// EN: Endpoint flags depend on actual feedback and remain valid
//     independently of the active automatic target.
// PT: As flags de extremidade dependem do feedback real e permanecem
//     válidas independentemente do alvo automático ativo.
elevatorAtMinPosition :=
    elevatorHomed AND
    (
        elevatorLowerLimit OR
        (
            elevatorPositionMm <=
            (
                machineConfig.elevatorMinPositionMm +
                MAX(0.0, machineConfig.elevatorPositionToleranceMm)
            )
        )
    );

elevatorAtMaxPosition :=
    elevatorHomed AND
    (
        elevatorUpperLimit OR
        (
            elevatorPositionMm >=
            (
                machineConfig.elevatorMaxPositionMm -
                MAX(0.0, machineConfig.elevatorPositionToleranceMm)
            )
        )
    );

elevatorInPosition :=
    elevatorHomed AND
    (
        (elevatorAbsPositionErrorMm <= machineConfig.elevatorPositionToleranceMm)
        OR
        (
            elevatorUpperLimit AND
            (elevatorTargetPositionMm >= machineConfig.elevatorMaxPositionMm)
        )
        OR
        (
            elevatorLowerLimit AND
            (elevatorTargetPositionMm <= machineConfig.elevatorMinPositionMm)
        )
    );


//==============================================================
// 5) Fault reset
//==============================================================
IF resetCmd AND
   safetyCircuitOk AND
   elevatorDriveOk AND
   NOT elevatorUpperSafetyLimit AND
   NOT elevatorLowerSafetyLimit THEN

    elevatorFault := FALSE;
    elevatorFaultCode := 0;

    IF elevatorControlState = 90 THEN
        elevatorControlState := 0;
    END_IF

END_IF;


//==============================================================
// 6) Invalidate an interrupted homing sequence
//==============================================================
// EN: If homing or its final upward movement is interrupted by a
//     protection/system stop, a new homing cycle is required.
// PT: Se o homing ou sua subida final for interrompido por proteção/parada,
//     um novo ciclo de homing será obrigatório.
IF (elevatorControlState >= 10) AND
   (elevatorControlState <= 14) AND
   (
       NOT systemRunEnable OR
       NOT safetyCircuitOk OR
       NOT elevatorDriveOk OR
       elevatorUpperSafetyLimit OR
       elevatorLowerSafetyLimit
   ) THEN

    elevatorHomed := FALSE;
    elevatorReadyForAutomaticCycle := FALSE;

END_IF;


//==============================================================
// 7) General protection
//==============================================================
IF NOT safetyCircuitOk THEN

    elevatorState := 'SAFETY_OFF';
    elevatorFault := TRUE;
    elevatorFaultCode := 2;
    elevatorControlState := 90;

    tonElevatorHomingTimeout(IN := FALSE);
    tonElevatorHomeSettleDelay(IN := FALSE);
    tonElevatorLevelingSpeed2Delay(IN := FALSE);


ELSIF NOT elevatorDriveOk THEN

    elevatorState := 'DRIVE_NOT_OK';
    elevatorFault := TRUE;
    elevatorFaultCode := 1;
    elevatorControlState := 90;

    tonElevatorHomingTimeout(IN := FALSE);
    tonElevatorHomeSettleDelay(IN := FALSE);
    tonElevatorLevelingSpeed2Delay(IN := FALSE);


ELSIF elevatorUpperSafetyLimit THEN

    elevatorState := 'UPPER_SAFE_LIMIT';
    elevatorFault := TRUE;
    elevatorFaultCode := 4;
    elevatorControlState := 90;

    tonElevatorHomingTimeout(IN := FALSE);
    tonElevatorHomeSettleDelay(IN := FALSE);
    tonElevatorLevelingSpeed2Delay(IN := FALSE);


ELSIF elevatorLowerSafetyLimit THEN

    elevatorState := 'LOWER_SAFE_LIMIT';
    elevatorFault := TRUE;
    elevatorFaultCode := 5;
    elevatorControlState := 90;

    tonElevatorHomingTimeout(IN := FALSE);
    tonElevatorHomeSettleDelay(IN := FALSE);
    tonElevatorLevelingSpeed2Delay(IN := FALSE);


ELSIF NOT systemRunEnable THEN

    elevatorState := 'SYSTEM_DISABLED';
    elevatorSignedSpeedRefMmps := 0.0;

    tonElevatorHomingTimeout(IN := FALSE);
    tonElevatorHomeSettleDelay(IN := FALSE);
    tonElevatorLevelingSpeed2Delay(IN := FALSE);

    IF elevatorControlState <> 90 THEN
        elevatorControlState := 0;
    END_IF


ELSE

    //==========================================================
    // 8) Mode selection
    //==========================================================
    // EN: A new home command is ignored while discharge is active/pending.
    // PT: Novo comando de home é ignorado durante descarte ativo/pendente.
    IF rElevatorHome AND
       NOT elevatorFault AND
       NOT sheetStackDischargeActive AND
       NOT sheetStackDischargePending THEN

        elevatorControlState := 10;

    END_IF;

    // EN: Discharge override blocks manual and leveling commands.
    // PT: Override de descarte bloqueia comandos manuais e nivelamento.
    IF elevatorTargetOverrideActive AND
       elevatorHomed AND
       (elevatorControlState <> 10) AND
       (elevatorControlState <> 11) AND
       (elevatorControlState <> 12) AND
       (elevatorControlState <> 13) AND
       (elevatorControlState <> 14) AND
       (elevatorControlState <> 90) THEN

        elevatorControlState := 40;

    END_IF;


    //==========================================================
    // 9) Elevator state machine
    //==========================================================
    CASE elevatorControlState OF

        0: // STOP
            elevatorState := 'STOP';

            tonElevatorHomingTimeout(IN := FALSE);
            tonElevatorHomeSettleDelay(IN := FALSE);
            tonElevatorLevelingSpeed2Delay(IN := FALSE);

            // EN: Manual movement is available with automatic mode off.
            //     With automatic mode on, it is available only after homing
            //     and completion of the upper home positioning.
            // PT: O movimento manual fica disponível com o automático desligado.
            //     Com o automático ligado, fica disponível somente após o homing
            //     e a conclusão do posicionamento superior.
            IF elevatorManualCommandRequest AND
               (
                   NOT elevatorAutoCmd OR
                   (
                       elevatorHomed AND
                       elevatorReadyForAutomaticCycle
                   )
               ) THEN

                elevatorControlState := 20;

            ELSIF elevatorAutoCmd AND
                  elevatorHomed AND
                  elevatorReadyForAutomaticCycle THEN

                elevatorControlState := 30;

            END_IF


        10: // HOME_DOWN_SEARCH
            elevatorState := 'HOME_DOWN';
            elevatorHomed := FALSE;
            elevatorReadyForAutomaticCycle := FALSE;
            elevatorInPosition := FALSE;

            tonElevatorHomingTimeout(
                IN := TRUE,
                PT := machineConfig.elevatorHomingTimeout
            );

            IF tonElevatorHomingTimeout.Q THEN

                elevatorSignedSpeedRefMmps := 0.0;
                tonElevatorHomingTimeout(IN := FALSE);

                elevatorFault := TRUE;
                elevatorFaultCode := 3;
                elevatorState := 'HOME_TIMEOUT';
                elevatorControlState := 90;

            ELSIF elevatorHomeLimitReached THEN

                elevatorSignedSpeedRefMmps := 0.0;
                tonElevatorHomingTimeout(IN := FALSE);
                elevatorControlState := 11;

            ELSIF elevatorHomeDownAllowed THEN

                elevatorSignedSpeedRefMmps :=
                    -ABS(machineConfig.elevatorHomingSpeedMmps);

            END_IF


        11: // HOME_RELEASE_SENSOR
            elevatorState := 'HOME_RELEASE';

            tonElevatorHomingTimeout(
                IN := TRUE,
                PT := machineConfig.elevatorHomingTimeout
            );

            IF tonElevatorHomingTimeout.Q THEN

                elevatorSignedSpeedRefMmps := 0.0;
                tonElevatorHomingTimeout(IN := FALSE);

                elevatorFault := TRUE;
                elevatorFaultCode := 3;
                elevatorState := 'HOME_TIMEOUT';
                elevatorControlState := 90;

            ELSIF elevatorHomeLimitFallingEdge THEN

                elevatorSignedSpeedRefMmps := 0.0;
                tonElevatorHomingTimeout(IN := FALSE);
                tonElevatorHomeSettleDelay(IN := FALSE);
                elevatorControlState := 12;

            ELSIF elevatorHomeReleaseAllowed THEN

                elevatorSignedSpeedRefMmps :=
                    ABS(machineConfig.elevatorHomingReleaseSpeedMmps);

            END_IF


        12: // HOME_SETTLE
            elevatorState := 'HOME_SETTLE';
            elevatorSignedSpeedRefMmps := 0.0;

            // EN: Encoder reset is allowed only while the lower sensor
            //     remains released throughout the settle time.
            // PT: Reset do encoder é permitido somente se o sensor inferior
            //     permanecer livre durante todo o tempo de estabilização.
            IF elevatorHomeLimitReached THEN

                tonElevatorHomeSettleDelay(IN := FALSE);
                elevatorControlState := 11;

            ELSE

                tonElevatorHomeSettleDelay(
                    IN := TRUE,
                    PT := machineConfig.elevatorHomeSettleDelay
                );

                IF tonElevatorHomeSettleDelay.Q THEN
                    tonElevatorHomeSettleDelay(IN := FALSE);
                    elevatorControlState := 13;
                END_IF

            END_IF


        13: // HOME_SET_ENCODER
            elevatorState := 'HOME_SET_ENCODER';
            elevatorSignedSpeedRefMmps := 0.0;

            elevatorSetEncoderPositionTrigger := TRUE;
            elevatorSetEncoderPositionMm := machineConfig.elevatorHomePositionMm;

            elevatorHomed := TRUE;
            elevatorFault := FALSE;
            elevatorFaultCode := 0;

            tonElevatorHomingTimeout(IN := FALSE);
            elevatorControlState := 14;


        14: // HOME_MOVE_TO_UPPER_POSITION
            elevatorState := 'HOME_MOVE_UP';

            tonElevatorHomingTimeout(
                IN := TRUE,
                PT := machineConfig.elevatorHomingTimeout
            );

            IF elevatorInPosition THEN

                elevatorSignedSpeedRefMmps := 0.0;
                tonElevatorHomingTimeout(IN := FALSE);
                elevatorReadyForAutomaticCycle := TRUE;

                IF elevatorAutoCmd THEN
                    elevatorControlState := 30;
                ELSE
                    elevatorControlState := 0;
                END_IF

            ELSIF tonElevatorHomingTimeout.Q THEN

                elevatorSignedSpeedRefMmps := 0.0;
                tonElevatorHomingTimeout(IN := FALSE);

                elevatorHomed := FALSE;
                elevatorReadyForAutomaticCycle := FALSE;
                elevatorFault := TRUE;
                elevatorFaultCode := 3;
                elevatorState := 'HOME_UP_TIMEOUT';
                elevatorControlState := 90;

            ELSIF (elevatorRawSpeedRefMmps > 0.0) AND elevatorUpAllowed THEN

                elevatorSignedSpeedRefMmps :=
                    elevatorRawSpeedRefMmps;

            ELSIF (elevatorRawSpeedRefMmps < 0.0) AND elevatorDownAllowed THEN

                elevatorSignedSpeedRefMmps :=
                    elevatorRawSpeedRefMmps;

            END_IF


        20: // MANUAL
            elevatorState := 'MANUAL';

            tonElevatorHomingTimeout(IN := FALSE);
            tonElevatorHomeSettleDelay(IN := FALSE);
            tonElevatorLevelingSpeed2Delay(IN := FALSE);

            // EN: Waiting for stack separation does not cancel manual operation.
            //     Active positioning or an elevator override cancels it.
            // PT: A espera pela separação da pilha não cancela a operação manual.
            //     O posicionamento ativo ou um override do elevador a cancela.
            IF sheetStackDischargeActive OR
               elevatorTargetOverrideActive THEN

                elevatorSignedSpeedRefMmps := 0.0;

                IF elevatorAutoCmd AND
                   elevatorHomed AND
                   elevatorReadyForAutomaticCycle THEN

                    elevatorControlState := 30;

                ELSE

                    elevatorControlState := 0;

                END_IF


            ELSIF elevatorAutoCmd AND
                  (
                      NOT elevatorHomed OR
                      NOT elevatorReadyForAutomaticCycle
                  ) THEN

                elevatorSignedSpeedRefMmps := 0.0;
                elevatorState := 'AUTO_NO_HOME';
                elevatorControlState := 0;

            ELSIF elevatorUpCmd AND elevatorDownCmd THEN

                elevatorSignedSpeedRefMmps := 0.0;

            ELSIF elevatorUpCmd THEN

                IF elevatorUpAllowed THEN

                    // EN: Reduce manual upward speed only while approaching
                    //     the configured maximum position.
                    // PT: Reduz a velocidade manual de subida somente durante
                    //     a aproximação da posição máxima configurada.
                    elevatorManualLowSpeedZoneActive :=
                        elevatorHomed AND
                        (
                            LIMIT(
                                0.0,
                                machineConfig.elevatorManualLowSpeedFactor,
                                1.0
                            ) < 1.0
                        ) AND
                        (
                            elevatorPositionMm >=
                            (
                                machineConfig.elevatorMaxPositionMm -
                                MAX(
                                    0.0,
                                    machineConfig.elevatorManualLowSpeedZoneMm
                                )
                            )
                        );

                    IF elevatorManualLowSpeedZoneActive THEN

                        elevatorSignedSpeedRefMmps :=
                            ABS(machineConfig.elevatorManualSpeedMmps) *
                            LIMIT(
                                0.0,
                                machineConfig.elevatorManualLowSpeedFactor,
                                1.0
                            );

                    ELSE

                        elevatorSignedSpeedRefMmps :=
                            ABS(machineConfig.elevatorManualSpeedMmps);

                    END_IF

                ELSE
                    elevatorSignedSpeedRefMmps := 0.0;
                END_IF

            ELSIF elevatorDownCmd THEN

                IF elevatorDownAllowed THEN

                    // EN: Reduce manual downward speed only while approaching
                    //     the configured minimum position.
                    // PT: Reduz a velocidade manual de descida somente durante
                    //     a aproximação da posição mínima configurada.
                    elevatorManualLowSpeedZoneActive :=
                        elevatorHomed AND
                        (
                            LIMIT(
                                0.0,
                                machineConfig.elevatorManualLowSpeedFactor,
                                1.0
                            ) < 1.0
                        ) AND
                        (
                            elevatorPositionMm <=
                            (
                                machineConfig.elevatorMinPositionMm +
                                MAX(
                                    0.0,
                                    machineConfig.elevatorManualLowSpeedZoneMm
                                )
                            )
                        );

                    IF elevatorManualLowSpeedZoneActive THEN

                        elevatorSignedSpeedRefMmps :=
                            -ABS(machineConfig.elevatorManualSpeedMmps) *
                            LIMIT(
                                0.0,
                                machineConfig.elevatorManualLowSpeedFactor,
                                1.0
                            );

                    ELSE

                        elevatorSignedSpeedRefMmps :=
                            -ABS(machineConfig.elevatorManualSpeedMmps);

                    END_IF

                ELSE
                    elevatorSignedSpeedRefMmps := 0.0;
                END_IF

            ELSE

                elevatorSignedSpeedRefMmps := 0.0;

                // EN: When manual intervention ends, automatic leveling
                //     may immediately evaluate the current level sensor.
                // PT: Ao terminar a intervenção manual, o nivelamento
                //     automático pode avaliar imediatamente o sensor atual.
                IF elevatorAutoCmd AND
                   elevatorHomed AND
                   elevatorReadyForAutomaticCycle THEN

                    elevatorControlState := 30;

                ELSE

                    elevatorControlState := 0;

                END_IF

            END_IF


        30: // AUTO_LEVELING
            elevatorState := 'AUTO_LEVELING';

            tonElevatorHomingTimeout(IN := FALSE);
            tonElevatorHomeSettleDelay(IN := FALSE);

            IF NOT elevatorAutoCmd THEN

                elevatorSignedSpeedRefMmps := 0.0;
                tonElevatorLevelingSpeed2Delay(IN := FALSE);
                elevatorControlState := 0;

            ELSIF NOT elevatorHomed OR
                  NOT elevatorReadyForAutomaticCycle THEN

                elevatorSignedSpeedRefMmps := 0.0;
                tonElevatorLevelingSpeed2Delay(IN := FALSE);
                elevatorState := 'AUTO_NO_HOME';

            ELSIF (elevatorUpCmd OR elevatorDownCmd) AND
                  NOT elevatorManualCommandArmed THEN

                // EN: A command held from homing or discharge inhibits
                //     leveling but cannot start a manual movement.
                // PT: Um comando mantido desde o homing ou descarte bloqueia
                //     o nivelamento, mas não pode iniciar movimento manual.
                elevatorSignedSpeedRefMmps := 0.0;
                tonElevatorLevelingSpeed2Delay(IN := FALSE);

            // EN: Manual correction remains available while the discharge
            //     sequence is waiting for stack separation.
            // PT: A correção manual permanece disponível enquanto a sequência
            //     de descarte aguarda a separação da pilha.
            ELSIF elevatorManualCommandRequest AND
                  NOT sheetStackDischargeActive AND
                  NOT elevatorTargetOverrideActive THEN

                // EN: Manual commands have priority over the level sensor.
                //     The speed-2 delay restarts after manual intervention.
                // PT: Os comandos manuais têm prioridade sobre o sensor de nível.
                //     O atraso da velocidade 2 reinicia após a intervenção manual.
                elevatorSignedSpeedRefMmps := 0.0;
                tonElevatorLevelingSpeed2Delay(IN := FALSE);
                elevatorControlState := 20;

            ELSIF backstopStackLevelSensor AND
                  elevatorDownAllowed THEN

                tonElevatorLevelingSpeed2Delay(
                    IN := TRUE,
                    PT := machineConfig.elevatorLevelingSpeed2Delay
                );

                IF tonElevatorLevelingSpeed2Delay.Q THEN
                    elevatorSignedSpeedRefMmps :=
                        -ABS(machineConfig.elevatorLevelingSpeed2Mmps);
                ELSE
                    elevatorSignedSpeedRefMmps :=
                        -ABS(machineConfig.elevatorLevelingSpeed1Mmps);
                END_IF

            ELSE

                elevatorSignedSpeedRefMmps := 0.0;
                tonElevatorLevelingSpeed2Delay(IN := FALSE);

            END_IF


        40: // DISCHARGE_POSITIONING
            elevatorState := 'DISCHARGE_POSITION';

            tonElevatorLevelingSpeed2Delay(IN := FALSE);

            IF NOT elevatorTargetOverrideActive THEN

                elevatorSignedSpeedRefMmps := 0.0;

                IF elevatorAutoCmd AND
                   elevatorHomed AND
                   elevatorReadyForAutomaticCycle THEN

                    elevatorControlState := 30;

                ELSE

                    elevatorControlState := 0;

                END_IF

            ELSIF elevatorInPosition THEN

                elevatorSignedSpeedRefMmps := 0.0;

            ELSIF (elevatorRawSpeedRefMmps > 0.0) AND elevatorUpAllowed THEN

                elevatorSignedSpeedRefMmps :=
                    elevatorRawSpeedRefMmps;

            ELSIF (elevatorRawSpeedRefMmps < 0.0) AND elevatorDownAllowed THEN

                elevatorSignedSpeedRefMmps :=
                    elevatorRawSpeedRefMmps;

            END_IF


        90: // FAULT
            elevatorState := 'FAULT';
            elevatorSignedSpeedRefMmps := 0.0;

            tonElevatorHomingTimeout(IN := FALSE);
            tonElevatorHomeSettleDelay(IN := FALSE);
            tonElevatorLevelingSpeed2Delay(IN := FALSE);


        ELSE
            elevatorControlState := 0;

    END_CASE;

END_IF;


//==============================================================
// 10) Encoder set pulse
//==============================================================
tpElevatorSetEncoderPosition(
    IN := elevatorSetEncoderPositionTrigger,
    PT := machineConfig.elevatorSetEncoderPulseTime
);

elevatorSetEncoderPosition := tpElevatorSetEncoderPosition.Q;


//==============================================================
// 11) Servo enable and magnetic brake control
//==============================================================
// EN: Keep the servo enabled with zero speed, following the backstop concept.
//     Drive-ready feedback is not used to avoid a circular enable dependency.
// PT: Mantém o servo habilitado com velocidade zero, seguindo o backstop.
//     O retorno de drive pronto não é usado para evitar dependência circular.
elevatorDriveEnable := systemRunEnable AND safetyCircuitOk;

elevatorMoveRequest :=
    systemRunEnable AND
    safetyCircuitOk AND
    elevatorDriveOk AND
    NOT elevatorFault AND
    (ABS(elevatorSignedSpeedRefMmps) > 0.0);

IF elevatorMoveRequest THEN

    elevatorBrakeReleaseRequest := TRUE;
    tonElevatorBrakeHoldDelay(IN := FALSE);

ELSE

    IF elevatorBrakeRelease THEN

        tonElevatorBrakeHoldDelay(
            IN := TRUE,
            PT := machineConfig.elevatorBrakeHoldTime
        );

        elevatorBrakeReleaseRequest :=
            NOT tonElevatorBrakeHoldDelay.Q;

    ELSE

        tonElevatorBrakeHoldDelay(IN := FALSE);
        elevatorBrakeReleaseRequest := FALSE;

    END_IF

END_IF;

elevatorBrakeRelease :=
    systemRunEnable AND
    safetyCircuitOk AND
    elevatorDriveOk AND
    NOT elevatorFault AND
    elevatorBrakeReleaseRequest;

tonElevatorBrakeReleaseDelay(
    IN := elevatorMoveRequest AND elevatorBrakeRelease,
    PT := machineConfig.elevatorBrakeReleaseDelay
);


//==============================================================
// 12) Direction and speed outputs
//==============================================================
IF elevatorMoveRequest AND
   elevatorBrakeRelease AND
   tonElevatorBrakeReleaseDelay.Q THEN

    elevatorSpeedRefMmps := elevatorSignedSpeedRefMmps;
    elevatorRunUp := elevatorSignedSpeedRefMmps > 0.0;
    elevatorRunDown := elevatorSignedSpeedRefMmps < 0.0;

ELSE

    elevatorSpeedRefMmps := 0.0;
    elevatorRunUp := FALSE;
    elevatorRunDown := FALSE;

END_IF;
END_METHOD

METHOD _ExternalCommands : BOOL
VAR_INPUT
END_VAR
END_METHOD

//==============================================================
// COMPLEX STACKER — HMI STATUS
// EN: Maps internal status, outputs, positions and diagnostics
//     to the HMI status structure.
//==============================================================
METHOD _HmiStatus



//==============================================================
// 1) System general status
//==============================================================
hmiStatus.systemRunEnable :=
    systemRunEnable;

hmiStatus.safetyCircuitOk :=
    safetyCircuitOk;

hmiStatus.faultActive :=
    faultActive OR
    (
        backstopRequiredForAutomaticOperation AND
        backstopFault
    ) OR
    elevatorFault OR
    sheetStackDischargeFault OR
    sheetStackDischargeConveyorFault;

hmiStatus.deviceState :=
    deviceState;


//==============================================================
// 2) Sheet conveyor group status
//==============================================================
hmiStatus.synchronizedConveyorsRunning :=
    synchronizedConveyorsRunning;

hmiStatus.sheetConveyor1Run :=
    sheetConveyor1Run;

hmiStatus.sheetConveyor2Run :=
    sheetConveyor2Run;

hmiStatus.sheetConveyor3Run :=
    sheetConveyor3Run;

hmiStatus.sheetConveyor4Run :=
    sheetConveyor4Run;

hmiStatus.sheetConveyor1SpeedRefMPM :=
    sheetConveyor1SpeedRefMPM;

hmiStatus.sheetConveyor2SpeedRefMPM :=
    sheetConveyor2SpeedRefMPM;

hmiStatus.sheetConveyor3SpeedRefMPM :=
    sheetConveyor3SpeedRefMPM;

hmiStatus.sheetConveyor4SpeedRefMPM :=
    sheetConveyor4SpeedRefMPM;

hmiStatus.syncConveyorsState :=
    syncConveyorsState;


//==============================================================
// 3) Sheet stack separation status
//==============================================================
hmiStatus.sheetStackSeparationReady :=
    sheetStackSeparationReady;

hmiStatus.sheetStackSeparationActive :=
    sheetStackSeparationActive;

hmiStatus.sheetStackBrakeActive :=
    sheetStackBrakeActive;


//==============================================================
// 4) Sheet stack discharge sequence status
//==============================================================
hmiStatus.sheetStackDischargeState :=
    sheetStackDischargeState;

hmiStatus.sheetStackDischargeStateCode :=
    sheetStackDischargeStateCode;

hmiStatus.sheetStackDischargePending :=
    sheetStackDischargePending;

hmiStatus.sheetStackDischargeActive :=
    sheetStackDischargeActive;

hmiStatus.sheetStackDischargeStarted :=
    sheetStackDischargeStarted;

hmiStatus.sheetStackDischargeFinished :=
    sheetStackDischargeFinished;

hmiStatus.sheetStackDischargeFault :=
    sheetStackDischargeFault;

hmiStatus.sheetStackDischargeFaultCode :=
    sheetStackDischargeFaultCode;

hmiStatus.sheetStackDischargeLastCycleOk :=
    sheetStackDischargeLastCycleOk;

hmiStatus.sheetStackDischargeLastResultCode :=
    sheetStackDischargeLastResultCode;

hmiStatus.sheetStackDischargeLastFaultStepCode :=
    sheetStackDischargeLastFaultStepCode;

hmiStatus.sheetStackDischargeLastFaultCode :=
    sheetStackDischargeLastFaultCode;


//==============================================================
// 5) Sheet stack discharge conveyor status
//==============================================================
hmiStatus.sheetStackDischargeConveyorState :=
    sheetStackDischargeConveyorState;

hmiStatus.sheetStackDischargeConveyorRun :=
    sheetStackDischargeConveyorRun;

hmiStatus.sheetStackDischargeConveyorSpeedRefMPM :=
    sheetStackDischargeConveyorSpeedRefMPM;

hmiStatus.sheetStackDischargeConveyorFault :=
    sheetStackDischargeConveyorFault;

hmiStatus.sheetStackDischargeConveyorFaultCode :=
    sheetStackDischargeConveyorFaultCode;


//==============================================================
// 6) Backstop status
//==============================================================
hmiStatus.backstopState :=
    backstopState;

hmiStatus.backstopHomed :=
    backstopHomed;

hmiStatus.backstopHomeRunning :=
    backstopHomeRunning;

hmiStatus.backstopInPosition :=
    backstopInPosition;

hmiStatus.backstopPositionMm :=
    backstopPositionMm;

hmiStatus.backstopTargetPositionMm :=
    backstopTargetPositionMm;

hmiStatus.backstopPositionErrorMm :=
    backstopPositionErrorMm;

hmiStatus.backstopRunFw :=
    backstopRunFw;

hmiStatus.backstopRunRev :=
    backstopRunRev;

hmiStatus.backstopSpeedRefMmps :=
    backstopSpeedRefMmps;

hmiStatus.backstopPlateUpSolenoid :=
    backstopPlateUpSolenoid;

hmiStatus.backstopSetEncoderPosition :=
    backstopSetEncoderPosition;

hmiStatus.backstopSetEncoderPositionMm :=
    backstopSetEncoderPositionMm;

hmiStatus.backstopManualInterventionActive :=
    backstopManualInterventionActive;

hmiStatus.backstopManualInterventionPositionMm :=
    backstopManualInterventionPositionMm;

hmiStatus.backstopFault :=
    backstopFault;

hmiStatus.backstopFaultCode :=
    backstopFaultCode;


//==============================================================
// 7) Elevator status
//==============================================================
hmiStatus.elevatorState :=
    elevatorState;

hmiStatus.elevatorHomed :=
    elevatorHomed;

hmiStatus.elevatorInPosition :=
    elevatorInPosition;

hmiStatus.elevatorPositionMm :=
    elevatorPositionMm;

hmiStatus.elevatorTargetPositionMm :=
    elevatorTargetPositionMm;

hmiStatus.elevatorPositionErrorMm :=
    elevatorPositionErrorMm;

hmiStatus.elevatorRunUp :=
    elevatorRunUp;

hmiStatus.elevatorRunDown :=
    elevatorRunDown;

hmiStatus.elevatorBrakeRelease :=
    elevatorBrakeRelease;

hmiStatus.elevatorSpeedRefMmps :=
    elevatorSpeedRefMmps;

hmiStatus.elevatorSetEncoderPosition :=
    elevatorSetEncoderPosition;

hmiStatus.elevatorSetEncoderPositionMm :=
    elevatorSetEncoderPositionMm;

hmiStatus.elevatorFault :=
    elevatorFault;

hmiStatus.elevatorFaultCode :=
    elevatorFaultCode;


//==============================================================
// 8) Process values
//==============================================================
hmiStatus.lineSpeedMPM :=
    lineSpeedMPM;

hmiStatus.sheetLengthMm :=
    sheetLengthMm;

hmiStatus.stackHeightMm :=
    stackHeightMm;


//==============================================================
// 9) Input / drive status mirror
//==============================================================
hmiStatus.sheetConveyor1DriveOk :=
    sheetConveyor1DriveOk;

hmiStatus.sheetConveyor2DriveOk :=
    sheetConveyor2DriveOk;

hmiStatus.sheetConveyor3DriveOk :=
    sheetConveyor3DriveOk;

hmiStatus.sheetConveyor4DriveOk :=
    sheetConveyor4DriveOk;

hmiStatus.backstopDriveOk :=
    backstopDriveOk;

hmiStatus.elevatorDriveOk :=
    elevatorDriveOk;

hmiStatus.sheetStackDischargeConveyorDriveOk :=
    sheetStackDischargeConveyorDriveOk;
END_METHOD

METHOD _MachineAuxilary
VAR_INPUT
END_VAR
(*



stopMachinePulse :=
    NOT safetyCircuitOk OR
    NOT sheetConveyor1DriveOk OR
    NOT sheetConveyor2DriveOk OR
    NOT sheetConveyor3DriveOk;
	NOT backstopDriveOk
	NOT elevatorDriveOk
*)
noCrushRollersUpDownValve := noCrushRollersDownCmd;

stackerRunning := systemRunEnable;


reset := resetCmd;
END_METHOD

//==============================================================
// COMPLEX STACKER — SHEET CONVEYOR GROUP CONTROL
// EN: Controls the synchronized sheet conveyor group.
//     Start/stop command latch is handled by _SystemControl().
//==============================================================
METHOD _SheetConveyorGroupControl

//==============================================================
// 1) Conditions
//==============================================================
// EN: Only synchronized sheet conveyor drives are considered here.
// PT: Apenas os inversores das esteiras sincronizadas são considerados aqui.
allSynchronizedDrivesOk :=
    sheetConveyor1DriveOk AND
    sheetConveyor2DriveOk AND
    sheetConveyor3DriveOk AND
    sheetConveyor4DriveOk;


// EN: Synchronized conveyor group fault.
// PT: Falha do grupo de esteiras sincronizadas.
anyFault :=
    NOT safetyCircuitOk OR
    NOT allSynchronizedDrivesOk;

faultActive := anyFault;


//==============================================================
// 2) State machine
//==============================================================
CASE syncConveyorsState OF

    0: // IDLE
        deviceState := 'IDLE';

        sheetConveyor1Run := FALSE;
        sheetConveyor2Run := FALSE;
        sheetConveyor3Run := FALSE;
        sheetConveyor4Run := FALSE;

        synchronizedConveyorsRunning := FALSE;

        // EN: The group starts only when the master system is enabled
        //     and no conveyor group fault is active.
        IF systemRunEnable AND NOT anyFault THEN

            syncConveyorsState := 1;

        ELSIF systemRunEnable AND anyFault THEN

            syncConveyorsState := 10;

        END_IF


    1: // RUN
        deviceState := 'RUN';

        // EN: Outputs are also directly conditioned by systemRunEnable
        //     to avoid one-scan movement after a stop command.
        sheetConveyor1Run :=
            systemRunEnable AND
            safetyCircuitOk AND
            sheetConveyor1DriveOk;

        sheetConveyor2Run :=
            systemRunEnable AND
            safetyCircuitOk AND
            sheetConveyor2DriveOk;

        sheetConveyor3Run :=
            systemRunEnable AND
            safetyCircuitOk AND
            sheetConveyor3DriveOk;

        sheetConveyor4Run :=
            systemRunEnable AND
            safetyCircuitOk AND
            sheetConveyor4DriveOk;

        synchronizedConveyorsRunning :=
            sheetConveyor1Run AND
            sheetConveyor2Run AND
            sheetConveyor3Run AND
            sheetConveyor4Run;

        IF anyFault THEN

            syncConveyorsState := 10;

        ELSIF NOT systemRunEnable THEN

            syncConveyorsState := 0;

        END_IF


    10: // FAULT
        deviceState := 'FAULT';

        sheetConveyor1Run := FALSE;
        sheetConveyor2Run := FALSE;
        sheetConveyor3Run := FALSE;
        sheetConveyor4Run := FALSE;

        synchronizedConveyorsRunning := FALSE;

        // EN: Fault state is released only by reset and with all faults cleared.
        //     If systemRunEnable is still TRUE after reset, the group can start
        //     again from IDLE on the next scan.
        IF resetCmd AND NOT anyFault THEN

            syncConveyorsState := 0;

        END_IF


ELSE

    syncConveyorsState := 0;

END_CASE;
END_METHOD

//==============================================================
// COMPLEX STACKER — SHEET STACK DISCHARGE CONTROL
// EN: Controls the sheet stack discharge sequence after the sheet
//     conveyor separation cycle is completed.
//
// State code
// 0  = IDLE
// 5  = WAIT_SEPARATION
// 10 = START_DISCHARGE_POSITIONING
// 20 = WAIT_DISCHARGE_POSITION
// 30 = RUN_DISCHARGE_CONVEYOR_AND_WAIT_CLEAR
// 40 = START_RETURN_POSITIONING
// 50 = WAIT_RETURN_POSITION
// 60 = FINISH
// 90 = FAULT_HOLD
//
// Last result code
// 0 = No cycle executed yet
// 1 = Last cycle completed successfully
// 2 = Last cycle completed with manual backstop skip
// 3 = Last cycle completed/aborted by timeout
// 4 = Last cycle aborted by fault
//
// Fault code
// 0  = No fault
// 1  = Safety circuit not OK
// 2  = Sheet conveyor drive not OK
// 3  = Discharge conveyor drive/control fault
// 4  = Backstop drive/control fault
// 5  = Elevator drive/control fault
// 6  = Stacker stopped during cycle
// 10 = Wait separation timeout
// 20 = Discharge positioning timeout
// 30 = Discharge conveyor did not start timeout
// 31 = Elevator platform clear timeout
// 50 = Return positioning timeout
//==============================================================
METHOD _SheetStackDischargeControl
VAR
    abortCycle : BOOL;
    backstopDischargeReady : BOOL;
    backstopAutomaticCycleEnabled : BOOL;
    elevatorPlatformClear : BOOL;
END_VAR


//==============================================================
// 1) Default event pulses
//==============================================================
sheetStackDischargeStarted  := FALSE;
sheetStackDischargeFinished := FALSE;

// EN: An empty platform is accepted even when no stack was present
//     at the beginning of the discharge cycle.
// PT: Plataforma vazia é aceita mesmo quando não havia pilha
//     no início do ciclo de descarte.
elevatorPlatformClear :=
    NOT elevatorStackPresentAtDischargeStart OR
    (
        elevatorStackExitClearSensor AND
        NOT elevatorStackPresentSensor
    );


//==============================================================
// 2) Default internal requests / overrides
//==============================================================
// EN: The sequence does not write the physical discharge conveyor outputs.
//     It only generates an internal request to the conveyor control method.
sheetStackDischargeConveyorRunRequest := FALSE;

backstopTargetOverrideActive := FALSE;
backstopTargetOverridePositionMm := 0.0;

elevatorTargetOverrideActive := FALSE;
elevatorTargetOverridePositionMm := 0.0;


//==============================================================
// 3) Edge detection
//==============================================================
// EN: Separate edge detector to avoid interfering with conveyor speed control.
rPackageCompleteDischarge :=
    packageCompleteCmd AND NOT packageCompleteCmdOldDischarge;

packageCompleteCmdOldDischarge := packageCompleteCmd;


//==============================================================
// 3.1) Backstop participation in the current cycle
//==============================================================
// EN: Once manual mode is detected during an accepted cycle, keep the
//     backstop bypassed until that cycle finishes. Returning the selector
//     to automatic cannot restart an old backstop movement.
// PT: Depois que o modo manual for detectado durante um ciclo aceito,
//     mantém o backstop ignorado até o fim desse ciclo. Retornar o seletor
//     para automático não reinicia um movimento antigo do backstop.
IF (
       sheetStackDischargeActive OR
       sheetStackDischargePending OR
       (sheetStackDischargeControlState <> 0)
   ) AND
   NOT backstopAutoCmd THEN

    sheetStackDischargeCycleHasManualSkip := TRUE;

END_IF;


IF sheetStackDischargeActive OR
   sheetStackDischargePending OR
   (sheetStackDischargeControlState <> 0) THEN

    backstopAutomaticCycleEnabled :=
        backstopAutoCmd AND
        NOT sheetStackDischargeCycleHasManualSkip;

ELSE

    // EN: Before accepting a new cycle, use the current selector position.
    // PT: Antes de aceitar um novo ciclo, usa a posição atual do seletor.
    backstopAutomaticCycleEnabled := backstopAutoCmd;

END_IF;


//==============================================================
// 4) Fault condition
//==============================================================
// EN: Elevator drive, homing and position feedback are required
//     for safe discharge sequence progress.
// PT: Drive, homing e posição do elevador são obrigatórios
//     para o avanço seguro da sequência de descarte.
sheetStackDischargeFaultCondition :=
    NOT safetyCircuitOk OR
    NOT sheetConveyor1DriveOk OR
    NOT sheetConveyor2DriveOk OR
    NOT sheetConveyor3DriveOk OR
    NOT sheetConveyor4DriveOk OR
    NOT sheetStackDischargeConveyorDriveOk OR
    sheetStackDischargeConveyorFault OR
    (
        backstopAutomaticCycleEnabled AND
        (
            NOT backstopDriveOk OR
            NOT backstopHomed OR
            backstopFault
        )
    ) OR
    NOT elevatorDriveOk OR
    NOT elevatorHomed OR
    NOT elevatorReadyForAutomaticCycle OR
    elevatorFault;


//==============================================================
// 5) Fault code priority
//==============================================================
IF NOT safetyCircuitOk THEN

    sheetStackDischargeFaultCode := 1;

ELSIF NOT sheetConveyor1DriveOk OR
      NOT sheetConveyor2DriveOk OR
      NOT sheetConveyor3DriveOk OR
      NOT sheetConveyor4DriveOk THEN

    sheetStackDischargeFaultCode := 2;

ELSIF NOT sheetStackDischargeConveyorDriveOk OR
      sheetStackDischargeConveyorFault THEN

    sheetStackDischargeFaultCode := 3;

ELSIF backstopAutomaticCycleEnabled AND
      (
          NOT backstopDriveOk OR
          NOT backstopHomed OR
          backstopFault
      ) THEN

    sheetStackDischargeFaultCode := 4;

ELSIF NOT elevatorDriveOk OR
      NOT elevatorHomed OR
      NOT elevatorReadyForAutomaticCycle OR
      elevatorFault THEN

    sheetStackDischargeFaultCode := 5;

ELSIF NOT synchronizedConveyorsRunning THEN

    sheetStackDischargeFaultCode := 6;

END_IF;


//==============================================================
// 6) Optional reset of current sequence fault display
//==============================================================
// EN: Reset clears the current sequence fault flag,
//     but does not erase last cycle diagnostic codes.
IF resetCmd AND (sheetStackDischargeControlState = 0) THEN

    sheetStackDischargeFault := FALSE;
    sheetStackDischargeFaultCode := 0;

END_IF;


//==============================================================
// 7) Arm discharge sequence from packageCompleteCmd
//==============================================================
// EN: packageCompleteCmd is ignored if the elevator is not in automatic,
//     the stacker is not running or a relevant drive/safety fault is active.
// PT: packageCompleteCmd é ignorado se o elevador não estiver em automático,
//     o stacker não estiver rodando ou houver falha relevante de drive/segurança.
IF rPackageCompleteDischarge AND
   elevatorAutoCmd AND
   synchronizedConveyorsRunning AND
   NOT sheetStackDischargeFaultCondition AND
   NOT sheetStackDischargeFault AND
   NOT sheetStackDischargeActive AND
   NOT sheetStackDischargePending THEN

    sheetStackDischargePending := TRUE;

    // EN: Clear current-cycle flags when a new cycle is accepted.
    sheetStackDischargeFault := FALSE;
    sheetStackDischargeFaultCode := 0;

    // EN: Manual is a valid bypass. It remains latched for this whole cycle.
    // PT: Manual é um bypass válido. Permanece memorizado por todo o ciclo.
    sheetStackDischargeCycleHasManualSkip := NOT backstopAutoCmd;
    sheetStackDischargeCycleHasTimeout := FALSE;

END_IF;


//==============================================================
// 8) Immediate abort condition
//==============================================================
// EN: Faults before discharge positioning cancel the request. Faults after
//     positioning starts hold safe targets until operator acknowledgement.
// PT: Falhas antes do posicionamento cancelam o pedido. Após o início,
//     mantêm os alvos seguros até o reconhecimento do operador.
abortCycle :=
    (
        sheetStackDischargeActive OR
        sheetStackDischargePending OR
        (sheetStackDischargeControlState <> 0)
    )
    AND
    (
        sheetStackDischargeFaultCondition OR
        NOT synchronizedConveyorsRunning
    );


IF abortCycle THEN

    sheetStackDischargeConveyorRunRequest := FALSE;
    sheetStackDischargePending := FALSE;

    tonSheetStackDischarge(IN := FALSE);
    tonSheetStackDischargeStepTimeout(IN := FALSE);
    tonSheetStackDischargePlatformClearTimeout(IN := FALSE);

    sheetStackDischargeFault := TRUE;

    sheetStackDischargeLastCycleOk := FALSE;
    sheetStackDischargeLastResultCode := 4;
    sheetStackDischargeLastFaultCode := sheetStackDischargeFaultCode;

    // EN: Do not clear backstopManualInterventionActive here.
    //     If the cycle aborted before return, keeping the memory is safer
    //     for the next cycle.

    IF sheetStackDischargeControlState <= 5 THEN

        // EN: No discharge movement has started yet.
        // PT: Nenhum movimento de descarte foi iniciado.
        sheetStackDischargeActive := FALSE;

        backstopTargetOverrideActive := FALSE;
        elevatorTargetOverrideActive := FALSE;

        elevatorPlatformClearDetected := FALSE;
        elevatorStackPresentAtDischargeStart := FALSE;

        sheetStackDischargeLastFaultStepCode :=
            sheetStackDischargeControlState;

        sheetStackDischargeState := 'ABORTED';
        sheetStackDischargeStateCode := 90;
        sheetStackDischargeControlState := 0;

    ELSE

        // EN: Preserve the original failed step while the external
        //     fault condition remains active in FAULT_HOLD.
        // PT: Preserva o passo original da falha enquanto a condição
        //     externa permanecer ativa no FAULT_HOLD.
        IF sheetStackDischargeControlState <> 90 THEN
            sheetStackDischargeLastFaultStepCode :=
                sheetStackDischargeControlState;
        END_IF;

        sheetStackDischargeActive := TRUE;
        sheetStackDischargeState := 'FAULT_HOLD';
        sheetStackDischargeStateCode := 90;

        IF sheetStackDischargeLastFaultStepCode < 40 THEN

            IF backstopAutomaticCycleEnabled THEN

                backstopTargetOverrideActive := TRUE;
                backstopTargetOverridePositionMm :=
                    backstopDischargeOpenTargetMm;

            END_IF;

            elevatorTargetOverrideActive := TRUE;
            elevatorTargetOverridePositionMm :=
                machineConfig.elevatorMinPositionMm;

        ELSE

            IF backstopAutomaticCycleEnabled THEN

                backstopTargetOverrideActive := TRUE;
                backstopTargetOverridePositionMm :=
                    backstopProgrammedDischargeTargetMm;

            END_IF;

            elevatorTargetOverrideActive := TRUE;
            elevatorTargetOverridePositionMm :=
                machineConfig.elevatorMaxPositionMm;

        END_IF;

        sheetStackDischargeControlState := 90;

    END_IF


ELSE

    //==============================================================
    // 9) Sheet stack discharge state machine
    //==============================================================
    CASE sheetStackDischargeControlState OF

        0: // IDLE
            sheetStackDischargeState := 'IDLE';
            sheetStackDischargeStateCode := 0;

            sheetStackDischargeActive := FALSE;

            sheetStackDischargeConveyorRunRequest := FALSE;

            backstopTargetOverrideActive := FALSE;
            elevatorTargetOverrideActive := FALSE;

            tonSheetStackDischarge(IN := FALSE);
            tonSheetStackDischargeStepTimeout(IN := FALSE);
            tonSheetStackDischargePlatformClearTimeout(IN := FALSE);
            elevatorPlatformClearDetected := FALSE;
            elevatorStackPresentAtDischargeStart := FALSE;

            IF sheetStackDischargePending THEN

                tonSheetStackDischarge(IN := FALSE);
                tonSheetStackDischargeStepTimeout(IN := FALSE);

                sheetStackDischargeControlState := 5;

            END_IF


        5: // WAIT_SEPARATION
            sheetStackDischargeState := 'WAIT_SEPARATION';
            sheetStackDischargeStateCode := 5;

            sheetStackDischargeActive := FALSE;

            sheetStackDischargeConveyorRunRequest := FALSE;

            backstopTargetOverrideActive := FALSE;
            elevatorTargetOverrideActive := FALSE;

            tonSheetStackDischarge(IN := FALSE);

            // EN: Wait for conveyor speed control to finish sheet stack separation.
            tonSheetStackDischargeStepTimeout(
                IN := TRUE,
                PT := machineConfig.sheetStackDischargeWaitSeparationTimeout
            );

            // EN: Complex stacker discharge starts only after conveyor 4
            //     completes the package separation sequence.
            // PT: O descarte do stacker complexo inicia somente depois que
            //     a esteira 4 concluir a sequência de separação do pacote.
            IF sheetStackSeparationFinished AND
               sheetConveyor4SeparationFinished THEN

                tonSheetStackDischargeStepTimeout(IN := FALSE);

                sheetStackDischargeControlState := 10;


            ELSIF tonSheetStackDischargeStepTimeout.Q THEN

                // EN: Separation did not finish. Do not discharge.
                tonSheetStackDischargeStepTimeout(IN := FALSE);

                sheetStackDischargePending := FALSE;
                sheetStackDischargeActive := FALSE;

                sheetStackDischargeFault := TRUE;
                sheetStackDischargeFaultCode := 10;

                sheetStackDischargeLastCycleOk := FALSE;
                sheetStackDischargeLastResultCode := 3;
                sheetStackDischargeLastFaultStepCode := 5;
                sheetStackDischargeLastFaultCode := 10;

                sheetStackDischargeControlState := 0;

            END_IF


        10: // START_DISCHARGE_POSITIONING
            sheetStackDischargeState := 'START_POSITIONING';
            sheetStackDischargeStateCode := 10;

            sheetStackDischargePending := FALSE;
            sheetStackDischargeActive := TRUE;
            sheetStackDischargeStarted := TRUE;

            elevatorPlatformClearDetected := FALSE;
            tonSheetStackDischargePlatformClearTimeout(IN := FALSE);
            elevatorStackPresentAtDischargeStart :=
                elevatorStackPresentSensor;

            tonSheetStackDischarge(IN := FALSE);
            tonSheetStackDischargeStepTimeout(IN := FALSE);

            //======================================================
            // EN: Latch programmed backstop target for this cycle.
            //     This is the normal position based on sheet length.
            //======================================================
            backstopProgrammedDischargeTargetMm :=
                LIMIT(
                    machineConfig.backstopMinPositionMm,
                    MAX(0.0, sheetLengthMm) +
                        machineConfig.backstopSheetLengthOffsetMm,
                    machineConfig.backstopMaxPositionMm
                );

            //======================================================
            // EN: Define safe opening base position.
            //
            // If the operator manually moved the backstop before the
            // automatic cycle, use the greater value between:
            // - programmed position
            // - last manual intervention position
            //
            // This prevents the automatic opening override from closing
            // the backstop onto the material.
            //
            // If there was no manual intervention, use only the programmed
            // position as the base.
            //======================================================
            IF backstopManualInterventionActive THEN

                backstopDischargeOpenBasePositionMm :=
                    MAX(
                        backstopProgrammedDischargeTargetMm,
                        backstopManualInterventionPositionMm
                    );

            ELSE

                backstopDischargeOpenBasePositionMm :=
                    backstopProgrammedDischargeTargetMm;

            END_IF;

            //======================================================
            // EN: Latch safe discharge open target.
            //     Offset is applied after selecting the safe base.
            //======================================================
            backstopDischargeOpenTargetMm :=
                LIMIT(
                    machineConfig.backstopMinPositionMm,
                    backstopDischargeOpenBasePositionMm +
                        machineConfig.backstopDischargeOpenOffsetMm,
                    machineConfig.backstopMaxPositionMm
                );

            // EN: Request safe backstop opening only when it participates
            //     in the current automatic cycle. Manual mode is bypassed.
            // PT: Solicita a abertura segura do backstop somente quando ele
            //     participa do ciclo automático atual. O modo manual é ignorado.
            IF backstopAutomaticCycleEnabled THEN

                backstopTargetOverrideActive := TRUE;
                backstopTargetOverridePositionMm :=
                    backstopDischargeOpenTargetMm;

            END_IF;

            // EN: Request the elevator lower discharge position.
            // PT: Solicita a posição inferior de descarte do elevador.
            elevatorTargetOverrideActive := TRUE;
            elevatorTargetOverridePositionMm :=
                machineConfig.elevatorMinPositionMm;

            sheetStackDischargeControlState := 20;


        20: // WAIT_DISCHARGE_POSITION
            sheetStackDischargeState := 'WAIT_DISCHARGE_POS';
            sheetStackDischargeStateCode := 20;

            sheetStackDischargeActive := TRUE;

            // EN: In manual mode do not command or wait for the backstop.
            // PT: No modo manual não comanda nem aguarda o backstop.
            IF backstopAutomaticCycleEnabled THEN

                backstopTargetOverrideActive := TRUE;
                backstopTargetOverridePositionMm :=
                    backstopDischargeOpenTargetMm;

                backstopDischargeReady := backstopInPosition;

            ELSE

                backstopTargetOverrideActive := FALSE;
                backstopDischargeReady := TRUE;

            END_IF;

            // EN: Keep the lower discharge target active and wait for feedback.
            // PT: Mantém o alvo inferior de descarte e aguarda o feedback.
            elevatorTargetOverrideActive := TRUE;
            elevatorTargetOverridePositionMm :=
                machineConfig.elevatorMinPositionMm;

            IF backstopDischargeReady AND elevatorInPosition THEN

                tonSheetStackDischargeStepTimeout(IN := FALSE);
                sheetStackDischargeControlState := 30;

            ELSE

                tonSheetStackDischargeStepTimeout(
                    IN := TRUE,
                    PT := machineConfig.sheetStackDischargePositioningTimeout
                );

                IF tonSheetStackDischargeStepTimeout.Q THEN

                    tonSheetStackDischargeStepTimeout(IN := FALSE);

                    sheetStackDischargeCycleHasTimeout := TRUE;
                    sheetStackDischargeFault := TRUE;
                    sheetStackDischargeFaultCode := 20;

                    sheetStackDischargeLastCycleOk := FALSE;
                    sheetStackDischargeLastResultCode := 3;
                    sheetStackDischargeLastFaultStepCode := 20;
                    sheetStackDischargeLastFaultCode := 20;

                    // EN: Do not start the discharge conveyor without
                    //     confirmed elevator positioning.
                    // PT: Não inicia a esteira de descarte sem confirmar
                    //     o posicionamento do elevador.
                    sheetStackDischargeControlState := 90;
                    sheetStackDischargeActive := TRUE;
                    sheetStackDischargePending := FALSE;

                END_IF

            END_IF


        30: // RUN_DISCHARGE_CONVEYOR
            sheetStackDischargeState := 'DISCHARGING';
            sheetStackDischargeStateCode := 30;

            sheetStackDischargeActive := TRUE;

            // EN: Keep the backstop open only if it participates in this cycle.
            // PT: Mantém o backstop aberto somente se ele participa deste ciclo.
            IF backstopAutomaticCycleEnabled THEN

                backstopTargetOverrideActive := TRUE;
                backstopTargetOverridePositionMm :=
                    backstopDischargeOpenTargetMm;

            END_IF;

            // EN: Keep elevator at the lower discharge position.
            // PT: Mantém o elevador na posição inferior de descarte.
            elevatorTargetOverrideActive := TRUE;
            elevatorTargetOverridePositionMm :=
                machineConfig.elevatorMinPositionMm;

            // EN: Request discharge conveyor run.
            //     Physical output is controlled by _SheetStackDischargeConveyorControl.
            sheetStackDischargeConveyorRunRequest := TRUE;

            // EN: If conveyor is not actually running, use start timeout.
            IF NOT sheetStackDischargeConveyorRun THEN

                tonSheetStackDischarge(IN := FALSE);
                tonSheetStackDischargePlatformClearTimeout(IN := FALSE);

                tonSheetStackDischargeStepTimeout(
                    IN := TRUE,
                    PT := machineConfig.sheetStackDischargeConveyorStartTimeout
                );

                IF tonSheetStackDischargeStepTimeout.Q THEN

                    // EN: Conveyor did not start. Do not stay trapped.
                    tonSheetStackDischargeStepTimeout(IN := FALSE);

                    sheetStackDischargeConveyorRunRequest := FALSE;

                    sheetStackDischargeCycleHasTimeout := TRUE;

                    sheetStackDischargeFault := TRUE;
                    sheetStackDischargeFaultCode := 30;

                    sheetStackDischargeLastCycleOk := FALSE;
                    sheetStackDischargeLastResultCode := 3;
                    sheetStackDischargeLastFaultStepCode := 30;
                    sheetStackDischargeLastFaultCode := 30;

                    sheetStackDischargeControlState := 90;

                END_IF


            ELSE

                // EN: Conveyor is running. Count minimum discharge time
                //     and wait for a clean elevator platform.
                // PT: A esteira está em movimento. Conta o tempo mínimo
                //     e aguarda a plataforma do elevador ficar livre.
                tonSheetStackDischargeStepTimeout(IN := FALSE);

                tonSheetStackDischarge(
                    IN := TRUE,
                    PT := machineConfig.sheetStackDischargeTime
                );

                IF elevatorPlatformClear THEN
                    elevatorPlatformClearDetected := TRUE;
                END_IF;

                tonSheetStackDischargePlatformClearTimeout(
                    IN := NOT elevatorPlatformClearDetected,
                    PT := machineConfig.sheetStackDischargePlatformClearTimeout
                );

                IF tonSheetStackDischarge.Q AND
                   elevatorPlatformClearDetected THEN

                    tonSheetStackDischarge(IN := FALSE);
                    tonSheetStackDischargePlatformClearTimeout(IN := FALSE);

                    sheetStackDischargeConveyorRunRequest := FALSE;

                    sheetStackDischargeControlState := 40;

                ELSIF tonSheetStackDischargePlatformClearTimeout.Q THEN

                    tonSheetStackDischarge(IN := FALSE);
                    tonSheetStackDischargePlatformClearTimeout(IN := FALSE);

                    sheetStackDischargeConveyorRunRequest := FALSE;

                    sheetStackDischargeCycleHasTimeout := TRUE;
                    sheetStackDischargeFault := TRUE;
                    sheetStackDischargeFaultCode := 31;

                    sheetStackDischargeLastCycleOk := FALSE;
                    sheetStackDischargeLastResultCode := 3;
                    sheetStackDischargeLastFaultStepCode := 30;
                    sheetStackDischargeLastFaultCode := 31;

                    // EN: Keep the elevator down and backstop open until reset.
                    // PT: Mantém o elevador embaixo e o backstop aberto até o reset.
                    sheetStackDischargeControlState := 90;

                END_IF

            END_IF


        40: // START_RETURN_POSITIONING
            sheetStackDischargeState := 'START_RETURN';
            sheetStackDischargeStateCode := 40;

            sheetStackDischargeActive := TRUE;

            sheetStackDischargeConveyorRunRequest := FALSE;

            tonSheetStackDischarge(IN := FALSE);
            tonSheetStackDischargeStepTimeout(IN := FALSE);

            // EN: Return the backstop only if it participates in this cycle.
            // PT: Retorna o backstop somente se ele participa deste ciclo.
            IF backstopAutomaticCycleEnabled THEN

                backstopTargetOverrideActive := TRUE;
                backstopTargetOverridePositionMm :=
                    backstopProgrammedDischargeTargetMm;

            END_IF;

            // EN: Request elevator return to the upper production position.
            // PT: Solicita o retorno do elevador à posição superior de produção.
            elevatorTargetOverrideActive := TRUE;
            elevatorTargetOverridePositionMm :=
                machineConfig.elevatorMaxPositionMm;

            sheetStackDischargeControlState := 50;


        50: // WAIT_RETURN_POSITION
            sheetStackDischargeState := 'WAIT_RETURN_POS';
            sheetStackDischargeStateCode := 50;

            sheetStackDischargeActive := TRUE;

            sheetStackDischargeConveyorRunRequest := FALSE;

            // EN: In manual mode do not command or wait for backstop return.
            // PT: No modo manual não comanda nem aguarda o retorno do backstop.
            IF backstopAutomaticCycleEnabled THEN

                backstopTargetOverrideActive := TRUE;
                backstopTargetOverridePositionMm :=
                    backstopProgrammedDischargeTargetMm;

                backstopDischargeReady := backstopInPosition;

            ELSE

                backstopTargetOverrideActive := FALSE;
                backstopDischargeReady := TRUE;

            END_IF;

            // EN: Keep the upper elevator target active and wait for feedback.
            // PT: Mantém o alvo superior do elevador e aguarda o feedback.
            elevatorTargetOverrideActive := TRUE;
            elevatorTargetOverridePositionMm :=
                machineConfig.elevatorMaxPositionMm;

            IF backstopDischargeReady AND elevatorInPosition THEN

                tonSheetStackDischargeStepTimeout(IN := FALSE);
                sheetStackDischargeControlState := 60;

            ELSE

                tonSheetStackDischargeStepTimeout(
                    IN := TRUE,
                    PT := machineConfig.sheetStackDischargeReturnTimeout
                );

                IF tonSheetStackDischargeStepTimeout.Q THEN

                    tonSheetStackDischargeStepTimeout(IN := FALSE);

                    sheetStackDischargeCycleHasTimeout := TRUE;
                    sheetStackDischargeFault := TRUE;
                    sheetStackDischargeFaultCode := 50;

                    sheetStackDischargeLastCycleOk := FALSE;
                    sheetStackDischargeLastResultCode := 3;
                    sheetStackDischargeLastFaultStepCode := 50;
                    sheetStackDischargeLastFaultCode := 50;

                    // EN: Do not report a completed cycle without confirmed
                    //     return positioning.
                    // PT: Não confirma o ciclo sem o posicionamento de retorno.
                    sheetStackDischargeActive := TRUE;
                    sheetStackDischargePending := FALSE;
                    sheetStackDischargeControlState := 90;

                END_IF

            END_IF


        90: // FAULT_HOLD
            sheetStackDischargeState := 'FAULT_HOLD';
            sheetStackDischargeStateCode := 90;

            sheetStackDischargeActive := TRUE;
            sheetStackDischargePending := FALSE;
            sheetStackDischargeConveyorRunRequest := FALSE;

            tonSheetStackDischarge(IN := FALSE);
            tonSheetStackDischargeStepTimeout(IN := FALSE);
            tonSheetStackDischargePlatformClearTimeout(IN := FALSE);

            // EN: Before platform clearance, keep the safe discharge
            //     positions: backstop open and elevator down.
            // PT: Antes da confirmação de plataforma livre, mantém as
            //     posições seguras: backstop aberto e elevador embaixo.
            IF sheetStackDischargeLastFaultStepCode < 40 THEN

                IF backstopAutomaticCycleEnabled THEN

                    backstopTargetOverrideActive := TRUE;
                    backstopTargetOverridePositionMm :=
                        backstopDischargeOpenTargetMm;

                END_IF;

                elevatorTargetOverrideActive := TRUE;
                elevatorTargetOverridePositionMm :=
                    machineConfig.elevatorMinPositionMm;

            ELSE

                // EN: A return-position timeout occurs only after the
                //     platform was confirmed clear. Keep the return targets.
                // PT: Timeout de retorno ocorre somente após confirmar a
                //     plataforma livre. Mantém os alvos de retorno.
                IF backstopAutomaticCycleEnabled THEN

                    backstopTargetOverrideActive := TRUE;
                    backstopTargetOverridePositionMm :=
                        backstopProgrammedDischargeTargetMm;

                END_IF;

                elevatorTargetOverrideActive := TRUE;
                elevatorTargetOverridePositionMm :=
                    machineConfig.elevatorMaxPositionMm;

            END_IF;

            // EN: Reset is an explicit operator acknowledgement.
            // PT: Reset é uma confirmação explícita do operador.
            IF resetCmd AND
               safetyCircuitOk AND
               (
                   NOT backstopAutomaticCycleEnabled OR
                   backstopDriveOk
               ) AND
               elevatorDriveOk AND
               (
                   elevatorPlatformClear OR
                   elevatorPlatformClearDetected OR
                   (sheetStackDischargeLastFaultStepCode >= 40)
               ) THEN

                sheetStackDischargeFault := FALSE;
                sheetStackDischargeFaultCode := 0;

                // EN: After acknowledgement, complete the automatic return
                //     instead of releasing production immediately.
                // PT: Após o reconhecimento, conclui o retorno automático
                //     antes de liberar novamente a produção.
                sheetStackDischargeControlState := 40;

            END_IF


        60: // FINISH
            sheetStackDischargeState := 'FINISH';
            sheetStackDischargeStateCode := 60;

            sheetStackDischargeActive := FALSE;
            sheetStackDischargePending := FALSE;
            sheetStackDischargeFinished := TRUE;

            sheetStackDischargeConveyorRunRequest := FALSE;

            backstopTargetOverrideActive := FALSE;
            elevatorTargetOverrideActive := FALSE;

            tonSheetStackDischarge(IN := FALSE);
            tonSheetStackDischargeStepTimeout(IN := FALSE);
            tonSheetStackDischargePlatformClearTimeout(IN := FALSE);
            elevatorPlatformClearDetected := FALSE;
            elevatorStackPresentAtDischargeStart := FALSE;

            IF sheetStackDischargeCycleHasTimeout THEN

                sheetStackDischargeLastCycleOk := FALSE;
                sheetStackDischargeLastResultCode := 3;

                // EN: Keep manual intervention memory after timeout.
                //     The backstop may not have returned correctly.

            ELSIF sheetStackDischargeCycleHasManualSkip THEN

                sheetStackDischargeLastCycleOk := FALSE;
                sheetStackDischargeLastResultCode := 2;
                sheetStackDischargeLastFaultStepCode := 0;
                sheetStackDischargeLastFaultCode := 0;

                sheetStackDischargeFault := FALSE;
                sheetStackDischargeFaultCode := 0;

                // EN: Keep manual intervention memory because the backstop
                //     was not controlled automatically.


            ELSE

                sheetStackDischargeLastCycleOk := TRUE;
                sheetStackDischargeLastResultCode := 1;
                sheetStackDischargeLastFaultStepCode := 0;
                sheetStackDischargeLastFaultCode := 0;

                sheetStackDischargeFault := FALSE;
                sheetStackDischargeFaultCode := 0;

                // EN: Cycle completed correctly and backstop returned to
                //     programmed target. Clear manual intervention memory.
                backstopManualInterventionActive := FALSE;
                backstopManualInterventionPositionMm := 0.0;

            END_IF

            // EN: Always return to IDLE automatically.
            sheetStackDischargeControlState := 0;


    ELSE

        sheetStackDischargeControlState := 0;

    END_CASE;

END_IF;
END_METHOD

//==============================================================
// COMPLEX STACKER — SHEET STACK DISCHARGE CONVEYOR CONTROL
// EN: Controls the sheet stack discharge conveyor.
//     Conveyor runs while manual button is pressed or while
//     automatic request is active and conveyor automatic mode is enabled.
//
// Fault code
// 0 = No fault
// 1 = Safety circuit not OK
// 2 = Discharge conveyor drive not OK
//==============================================================
METHOD _SheetStackDischargeConveyorControl
VAR
    manualRunRequest   : BOOL;
    automaticRunRequest: BOOL;
    finalRunRequest    : BOOL;
END_VAR
//==============================================================
// COMPLEX STACKER — SHEET STACK DISCHARGE CONVEYOR CONTROL
// EN: Controls the sheet stack discharge conveyor in manual pulse
//     or automatic sequence request.
//==============================================================


//==============================================================
// 1) Default outputs
//==============================================================
sheetStackDischargeConveyorRun := FALSE;
sheetStackDischargeConveyorSpeedRefMPM := 0.0;


//==============================================================
// 2) Run request selection
//==============================================================
// EN: Manual command is momentary. Conveyor runs while button is pressed.
manualRunRequest :=
    sheetStackDischargeConveyorManualRunCmd;


// EN: Automatic request is generated by the discharge sequence.
//     This conveyor is assumed to be available for automatic cycle
//     whenever the master system is enabled.
automaticRunRequest :=
    sheetStackDischargeConveyorRunRequest;


// EN: Master system enable blocks both manual and automatic movement.
finalRunRequest :=
    systemRunEnable AND
    (
        manualRunRequest OR
        automaticRunRequest OR
		backstopHomeRunning
    );


//==============================================================
// 3) Fault detection
//==============================================================
IF NOT safetyCircuitOk THEN

    sheetStackDischargeConveyorState := 'SAFETY_OFF';

    sheetStackDischargeConveyorFault := TRUE;
    sheetStackDischargeConveyorFaultCode := 1;


ELSIF NOT sheetStackDischargeConveyorDriveOk THEN

    sheetStackDischargeConveyorState := 'DRIVE_NOT_OK';

    sheetStackDischargeConveyorFault := TRUE;
    sheetStackDischargeConveyorFaultCode := 2;


ELSE

    //==============================================================
    // 4) Fault reset
    //==============================================================
    IF resetCmd THEN

        sheetStackDischargeConveyorFault := FALSE;
        sheetStackDischargeConveyorFaultCode := 0;

    END_IF;


    //==============================================================
    // 5) Conveyor output control
    //==============================================================
    IF sheetStackDischargeConveyorFault THEN

        sheetStackDischargeConveyorState := 'FAULT';

        sheetStackDischargeConveyorRun := FALSE;
        sheetStackDischargeConveyorSpeedRefMPM := 0.0;


    ELSIF NOT systemRunEnable THEN

        // EN: Master stop disables movement without generating a conveyor fault.
        sheetStackDischargeConveyorState := 'SYSTEM_DISABLED';

        sheetStackDischargeConveyorRun := FALSE;
        sheetStackDischargeConveyorSpeedRefMPM := 0.0;


    ELSIF finalRunRequest THEN

        IF automaticRunRequest THEN

            sheetStackDischargeConveyorState := 'AUTO_RUN';

        ELSE

            sheetStackDischargeConveyorState := 'MANUAL_RUN';

        END_IF;

        sheetStackDischargeConveyorRun := TRUE;

        sheetStackDischargeConveyorSpeedRefMPM :=
            LIMIT(
                0.0,
                machineConfig.sheetStackDischargeConveyorSpeedMPM,
                machineConfig.maximumSpeedMPM
            );


    ELSE

        sheetStackDischargeConveyorState := 'STOP';

        sheetStackDischargeConveyorRun := FALSE;
        sheetStackDischargeConveyorSpeedRefMPM := 0.0;

    END_IF

END_IF;
END_METHOD

//==============================================================
// COMPLEX STACKER - STACK BUFFER CONVEYOR CONTROL
// EN: Transfers finished stacks to the furthest available buffer.
// PT: Transfere as pilhas prontas para o buffer livre mais distante.
//==============================================================
METHOD _StackBufferConveyorsControl
VAR
    allBufferDrivesOk : BOOL;
    automaticTransferActive : BOOL;
END_VAR
//==============================================================
// 1) Common conditions and edge detection
//==============================================================
allBufferDrivesOk :=
    stackBufferConveyor1DriveOk AND
    stackBufferConveyor2DriveOk AND
    stackBufferConveyor3DriveOk;

stackBufferFull :=
    stackBufferConveyor1StackPresentSensor AND
    stackBufferConveyor2StackPresentSensor AND
    stackBufferConveyor3StackPresentSensor;

rElevatorStackExitClear :=
    elevatorStackExitClearSensor AND
    NOT elevatorStackExitClearSensorOld;

elevatorStackExitClearSensorOld := elevatorStackExitClearSensor;

tonStackBufferFullSpeedReduction(
    IN := stackBufferFull,
    PT := machineConfig.stackBufferFullSpeedReductionDelay
);

lineSpeedReductionRequest := tonStackBufferFullSpeedReduction.Q;


//==============================================================
// 2) Default outputs
//==============================================================
stackBufferConveyor1Run := FALSE;
stackBufferConveyor2Run := FALSE;
stackBufferConveyor3Run := FALSE;

stackBufferConveyor1SpeedRefMPM := 0.0;
stackBufferConveyor2SpeedRefMPM := 0.0;
stackBufferConveyor3SpeedRefMPM := 0.0;


//==============================================================
// 3) Manual operation
// EN: Manual command ignores the stack presence sensors, but continues
//     to respect the master enable, safety circuit and drive status.
// PT: O comando manual ignora os sensores de presença, mas continua
//     respeitando a habilitação geral, segurança e estado dos drives.
//==============================================================
IF stackBufferConveyorsRunCmd THEN

    stackBufferControlState := 0;
    stackBufferTargetConveyor := 0;

    tonStackBufferStopDelay(IN := FALSE);
    tonStackBufferTransferTimeout(IN := FALSE);

    IF systemRunEnable AND safetyCircuitOk AND allBufferDrivesOk THEN

        stackBufferConveyor1Run := TRUE;
        stackBufferConveyor2Run := TRUE;
        stackBufferConveyor3Run := TRUE;

    END_IF


//==============================================================
// 4) Automatic accumulation
//==============================================================
ELSE

    // EN: A full buffer blocks automatic transfer and stops all conveyors.
    // PT: Buffer cheio bloqueia a transferência automática e para as esteiras.
    IF stackBufferFull OR
       NOT systemRunEnable OR
       NOT safetyCircuitOk OR
       NOT allBufferDrivesOk THEN

        stackBufferControlState := 0;
        stackBufferTargetConveyor := 0;

        tonStackBufferStopDelay(IN := FALSE);
        tonStackBufferTransferTimeout(IN := FALSE);

    ELSE

        CASE stackBufferControlState OF

            0: // IDLE
                tonStackBufferStopDelay(IN := FALSE);
                tonStackBufferTransferTimeout(IN := FALSE);

                IF rElevatorStackExitClear THEN

                    // EN: Always select the furthest available position.
                    // PT: Seleciona sempre a posição livre mais distante.
                    IF NOT stackBufferConveyor3StackPresentSensor THEN
                        stackBufferTargetConveyor := 3;
                        stackBufferControlState := 30;

                    ELSIF NOT stackBufferConveyor2StackPresentSensor THEN
                        stackBufferTargetConveyor := 2;
                        stackBufferControlState := 20;

                    ELSIF NOT stackBufferConveyor1StackPresentSensor THEN
                        stackBufferTargetConveyor := 1;
                        stackBufferControlState := 10;

                    END_IF

                END_IF


            10: // TRANSFER TO BUFFER 1
                stackBufferConveyor1Run := TRUE;

                IF stackBufferConveyor1StackPresentSensor THEN
                    tonStackBufferStopDelay(IN := FALSE);
                    stackBufferControlState := 11;
                END_IF


            11: // BUFFER 1 STOP DELAY
                stackBufferConveyor1Run := TRUE;

                tonStackBufferStopDelay(
                    IN := TRUE,
                    PT := machineConfig.stackBufferConveyorsStopDelay
                );

                IF tonStackBufferStopDelay.Q THEN
                    tonStackBufferStopDelay(IN := FALSE);
                    stackBufferControlState := 0;
                    stackBufferTargetConveyor := 0;
                END_IF


            20: // TRANSFER TO BUFFER 2
                stackBufferConveyor1Run := TRUE;
                stackBufferConveyor2Run := TRUE;

                IF stackBufferConveyor2StackPresentSensor THEN
                    tonStackBufferStopDelay(IN := FALSE);
                    stackBufferControlState := 21;
                END_IF


            21: // BUFFER 2 STOP DELAY
                stackBufferConveyor1Run := TRUE;
                stackBufferConveyor2Run := TRUE;

                tonStackBufferStopDelay(
                    IN := TRUE,
                    PT := machineConfig.stackBufferConveyorsStopDelay
                );

                IF tonStackBufferStopDelay.Q THEN
                    tonStackBufferStopDelay(IN := FALSE);
                    stackBufferControlState := 0;
                    stackBufferTargetConveyor := 0;
                END_IF


            30: // TRANSFER TO BUFFER 3
                stackBufferConveyor1Run := TRUE;
                stackBufferConveyor2Run := TRUE;
                stackBufferConveyor3Run := TRUE;

                // EN: Conveyor 3 stops immediately when its sensor is active.
                // PT: A esteira 3 para imediatamente quando seu sensor é acionado.
                IF stackBufferConveyor3StackPresentSensor THEN
                    stackBufferConveyor1Run := FALSE;
                    stackBufferConveyor2Run := FALSE;
                    stackBufferConveyor3Run := FALSE;

                    stackBufferControlState := 0;
                    stackBufferTargetConveyor := 0;
                END_IF


            ELSE
                stackBufferControlState := 0;
                stackBufferTargetConveyor := 0;

        END_CASE


        //==========================================================
        // 5) Automatic transfer timeout
        //==========================================================
        automaticTransferActive :=
            (stackBufferControlState <> 0);

        tonStackBufferTransferTimeout(
            IN := automaticTransferActive,
            PT := machineConfig.stackBufferTransferTimeout
        );

        IF tonStackBufferTransferTimeout.Q THEN
            tonStackBufferTransferTimeout(IN := FALSE);
            tonStackBufferStopDelay(IN := FALSE);

            stackBufferControlState := 0;
            stackBufferTargetConveyor := 0;

            stackBufferConveyor1Run := FALSE;
            stackBufferConveyor2Run := FALSE;
            stackBufferConveyor3Run := FALSE;
        END_IF

    END_IF

END_IF


//==============================================================
// 6) Apply the common fixed speed reference
//==============================================================
IF stackBufferConveyor1Run THEN
    stackBufferConveyor1SpeedRefMPM :=
        machineConfig.stackBufferConveyorsSpeedMPM;
END_IF;

IF stackBufferConveyor2Run THEN
    stackBufferConveyor2SpeedRefMPM :=
        machineConfig.stackBufferConveyorsSpeedMPM;
END_IF;

IF stackBufferConveyor3Run THEN
    stackBufferConveyor3SpeedRefMPM :=
        machineConfig.stackBufferConveyorsSpeedMPM;
END_IF;
END_METHOD

//==============================================================
// COMPLEX STACKER — SYSTEM CONTROL
// EN: Master system run enable and automatic homing requests.
//==============================================================
METHOD _SystemControl

//==============================================================
// 1) Edge detection
//==============================================================
rStartCmd := startCmd AND NOT startCmdOld;
startCmdOld := startCmd;

rStopCmd := stopCmd AND NOT stopCmdOld;
stopCmdOld := stopCmd;



//==============================================================
// 2) Stop machine pulse on critical fault
//==============================================================
// EN: A backstop bypassed in manual remains ignored until the current
//     discharge cycle finishes, even if the selector returns to automatic.
// PT: Um backstop ignorado em manual permanece fora do ciclo até o descarte
//     atual terminar, mesmo que o seletor retorne para automático.
backstopRequiredForAutomaticOperation :=
    backstopAutoCmd AND
    NOT (
        sheetStackDischargeCycleHasManualSkip AND
        (
            sheetStackDischargeActive OR
            sheetStackDischargePending OR
            (sheetStackDischargeControlState <> 0)
        )
    );


stopMachineFaultCondition :=
    NOT safetyCircuitOk OR
    NOT sheetConveyor1DriveOk OR
    NOT sheetConveyor2DriveOk OR
    NOT sheetConveyor3DriveOk OR
    NOT sheetConveyor4DriveOk OR
    (
        backstopRequiredForAutomaticOperation AND
        NOT backstopDriveOk
    ) OR
    NOT elevatorDriveOk OR
    NOT sheetStackDischargeConveyorDriveOk;

rStopMachineFaultCondition :=
    stopMachineFaultCondition AND
    NOT stopMachineFaultConditionOld;

stopMachineFaultConditionOld :=
    stopMachineFaultCondition;

tpStopMachinePulse(
    IN := rStopMachineFaultCondition,
    PT := T#500MS
);

stopMachinePulse :=
    tpStopMachinePulse.Q;


//==============================================================
// 2) Default one-scan requests
//==============================================================
backstopAutoHomeRequest := FALSE;
elevatorAutoHomeRequest := FALSE;


//==============================================================
// 3) Master system run enable
//==============================================================
IF NOT safetyCircuitOk THEN

    systemRunEnable := FALSE;

ELSIF rStopCmd THEN

    systemRunEnable := FALSE;

ELSIF rStartCmd THEN

    systemRunEnable := TRUE;

END_IF;


//==============================================================
// 4) Automatic homing on system start
//==============================================================
// EN: Auto-home is generated only on the rising edge of startCmd.
//     Each axis must be enabled in automatic mode.
//     This prevents automatic movement of axes intentionally left in manual.
IF rStartCmd AND systemRunEnable THEN

    // Backstop auto-home
    IF backstopAutoCmd AND
       NOT backstopHomed AND
       NOT backstopFault THEN

        backstopAutoHomeRequest := TRUE;

    END_IF;


    // Elevator auto-home
    IF elevatorAutoCmd AND
       NOT elevatorHomed AND
       NOT elevatorFault THEN

        elevatorAutoHomeRequest := TRUE;

    END_IF;

END_IF;
END_METHOD

END_FUNCTION_BLOCK

(* stored: Version 1.1.0.1
   POU FB_ComplexSheetStackerControl: Id {48f3d714-da40-448b-b8a6-71c59012c754}, SpecialFunc None
   Method _AlarmControl: Id {45013390-3a2e-451c-bcaa-d7957f4db2e9}
   Method _BackstopControl: Id {a8131784-f5c8-4a18-af8b-160d5c9efcab}
   Method _ConveyorSpeedControl: Id {b62cf8f8-3272-4eb3-b76e-d7c96032c01b}
   Method _ElevatorControl: Id {02ae8aac-d808-47f5-84f8-70101e7732c2}
   Method _ExternalCommands: Id {2305ba90-1f64-48e0-803d-b7af95d3af82}
   Method _HmiStatus: Id {9f9c3433-b925-4b5b-a55b-93a1136a64ce}
   Method _MachineAuxilary: Id {737ee558-6100-438a-96e5-47721d84e85a}
   Method _SheetConveyorGroupControl: Id {f14f5fe3-bf14-462b-8073-c7cc7907504e}
   Method _SheetStackDischargeControl: Id {6a21452b-a00c-4dc6-803c-d98058ed2a21}
   Method _SheetStackDischargeConveyorControl: Id {596c6d49-7c22-4b2d-ab6c-e3bef636eaa1}
   Method _StackBufferConveyorsControl: Id {63bd4e07-85e3-4f24-8234-299460111c67}
   Method _SystemControl: Id {f2b38b6a-adbc-4897-aa71-724486624911} *)
